{attribute addProperty BoxType "EL5032-0000-0021"}
{attribute addProperty Id "FB_Inputs_ChannelAT %I*ARRAY[0..1] OF FB_Inputs_Channel_FFB44ACB160200WcStateAT %I*WcState_98A4DF7520.250InfoDataAT %I*InfoData_BC63D37F80100"}
{attribute addProperty CRC "3319135795"}
{attribute addProperty SizeInBites "242"}
{attribute addProperty SizeInBytes "30.25"}
TYPE EL5032_3D8BD04C :
STRUCT
	{attribute addProperty Name "FB_Inputs_Channel"}
	FB_Inputs_Channel : ARRAY[0..1] OF FB_Inputs_Channel_FFB44ACB;
	{attribute addProperty Name "WcState"}
	WcState : WcState_98A4DF75;
	{attribute addProperty Name "InfoData"}
	InfoData : InfoData_BC63D37F;
END_STRUCT
END_TYPE

(* stored: Version 1.2.0.0, ProductVersion 3.1.4024.9
   DUT EL5032_3D8BD04C: Id {139eb302-8023-4402-bb6d-761b9227521a} *)
